// TwinCAT 3 PLC project Untitled1
// ProgramVersion: 3.1.4024.0
// libraries:
//   JSC_MC_Lib, * (Jenny Science AG)
//   JS_MC_REF, * (Jenny Science AG)
//   Sei_Standard, * (Sorenson Engineering)
//   Tc2_MC2, * (Beckhoff Automation GmbH)
//   Tc2_Standard, * (Beckhoff Automation GmbH)
//   Tc2_System, * (Beckhoff Automation GmbH)
//   Tc3_EventLogger, * (Beckhoff Automation GmbH)
//   Tc3_Module, * (Beckhoff Automation GmbH)
// project tree:
//   DUTs/ E_CIM_ERROR_CODES.TcDUT, ST_CONTACT_AFS_PARAMS.TcDUT, ST_CYCLE_TRACKING.TcDUT, ST_ERROR_LOG.TcDUT, ST_JOB_INFO.TcDUT, ST_PLACEMENT_DATA.TcDUT, ST_PLACEMENT_ERROR_INFO.TcDUT, ST_PRODUCTION_DATA.TcDUT, ST_RECIPE_VARS.TcDUT, ST_RFID_DATA.TcDUT, ST_SEARCH_SHAPE.TcDUT
//   GVLs/ GVL.TcGVL
//   ITFs/ ITF_Error.TcIO
//   / PlcTask.TcTTO
//   POUs/00_Shared/ FB_AlarmListener.TcPOU
//   POUs/ FB_AxisBase.TcPOU, FB_Button.TcPOU, FB_Light.TcPOU, FB_Motor.TcPOU, FB_XenaxAxisForceFeedback.TcPOU, MAIN.TcPOU
// real-time tasks:
//   TASK PlcTask: cycle T#10ms, priority 20, ADS port 350
// motion (NC):
//   TASK NC-Task 1 SAF: cycle T#1ms, priority 4, ADS port 501
//   TASK NC-Task 1 SVB: cycle T#10ms, priority 8, ADS port 511
//   AXIS Axis 1 (id 1)
//     General: UnitName=Degree
//     Dynamic: Acceleration=12748, Deceleration=500000, Jerk=382440
//     Velo: RefSync=50, SlowManual=90, FastManual=500, Fast=8498, Maximum=14400
//     PositionAreaControl: Enable=false
//     TargetPosControl: Enable=false
//     OtherSettings: AllowMotionCmdToSlave=true
//     encoder EncType=19
//       EncPara: ScaleFactorNumerator=360, ScaleFactorDenominator=120000, MaxCount=#xffffffff
//         SoftEndMinControl: Range=-29
//         SoftEndMaxControl: Range=29
//     drive DrvType=16
//       DrvPara: MaxCount=#xffffffff, DriveControlDWord=#x00000100
//         Analog: VeloReferenz=14400, VeloScale=32, TorqueSetpointScale=10, ScaleFactorActTorque=0.1
//         TimeComp: TaskDelayCycles=1
//     controller CtrType=9
//       CtrPara: PriorControlFactor=1
//         PosDiffControl: Enable=false, Range=8
//         Observer: BandWidth=20
// I/O:
//   DEVICE Device 2 (EtherCAT), AmsNetId 169.254.194.147.3.1
//     Term 6 (EK1100) [EK1100 EtherCAT Coupler (2A E-Bus)]
//       Term 7 (EL3174) [EL3174 4Ch. Ana. Input +/-10V Diff., +/-20mA SingleEnded, 16 Bit]
//       Term 8 (EL2828) [EL2828 8Ch. Dig. Output 24V, 2A]
//       Term 9 (EL6224) [EL6224 (IO Link Master)]
//       Term 11 (EL9011) [EL9011 End Terminal]
//     Drive 10 (Xvi) [XENAX Xvi 48V8]
// variable links:
//   NC-Task 1 SAF/Axes/Axis 1 <-> Device 2 (EtherCAT)/Drive 10 (Xvi)
//     Drive/Inputs/In/nDataIn1 <-> TxPDO 1/Following Error Actual Value
//     Drive/Inputs/In/nState1 <-> TxPDO 1/Statusword
//     Drive/Inputs/In/nState2 <-> TxPDO 1/Statusword @bit 8
//     Drive/Inputs/In/nState4 @bit 1 <-> WcState/InputToggle
//     Drive/Inputs/In/nState4 <-> WcState/WcState
//     Drive/Outputs/Out/nCtrl1 <-> RxPDO 1/Controlword
//     Drive/Outputs/Out/nCtrl2 <-> RxPDO 1/Controlword @bit 8
//     Drive/Outputs/Out/nDataOut1 <-> RxPDO 1/Target Position
//     Enc/Inputs/In/nDataIn1 <-> TxPDO 1/Position Actual Value
//     Enc/Inputs/In/nState4 @bit 1 <-> WcState/InputToggle
//     Enc/Inputs/In/nState4 <-> WcState/WcState
//   Untitled1/Untitled1 Instance <-> Device 2 (EtherCAT)/Drive 10 (Xvi)
//     PlcTask Inputs/MAIN.motor.ThisMotor.instJS_MC_Init.RxPDO/bWcState <-> WcState/WcState
//     PlcTask Inputs/MAIN.motor.ThisMotor.instJS_MC_Init.RxPDO/diProcessStatusRegister_I2006 <-> TxPDO 2/Process Status Register
//     PlcTask Inputs/MAIN.motor.ThisMotor.instJS_MC_Init.RxPDO/uiStatusword_I6041 <-> TxPDO 2/Statusword
//     PlcTask Inputs/MAIN.motor.ThisMotor.instJS_MC_Init.stSlaveAmsAddr/netId <-> InfoData/AdsAddr/netId
//     PlcTask Inputs/MAIN.motor.ThisMotor.instJS_MC_Init.stSlaveAmsAddr/port <-> InfoData/AdsAddr/port
//   Untitled1/Untitled1 Instance <-> Device 2 (EtherCAT)/Term 6 (EK1100)/Term 9 (EL6224)
//     PlcTask Inputs/MAIN.motor.button.byButtonInput <-> IO-Link Port2/Port2: process data
//     PlcTask Outputs/MAIN.motor.button.byButtonLight <-> IO-Link Port3/Port3: process data
//     PlcTask Outputs/MAIN.motor.light.bAnimationMode <-> IO-Link Port1/Animation Type
//     PlcTask Outputs/MAIN.motor.light.bColor1 <-> IO-Link Port1/Color 1
//     PlcTask Outputs/MAIN.motor.light.bColor2 <-> IO-Link Port1/Color 2
//     PlcTask Outputs/MAIN.motor.light.bColor1Intensity <-> IO-Link Port1/Color 1 Intensity
//     PlcTask Outputs/MAIN.motor.light.bColor2Intensity <-> IO-Link Port1/Color 2 Intensity
//     PlcTask Outputs/MAIN.motor.light.bFlashRate <-> IO-Link Port1/Color Flash Rate (Hz)
//     PlcTask Outputs/MAIN.motor.light.bRotationalMode <-> IO-Link Port1/Rotation Direction
//   Untitled1/Untitled1 Instance <-> NC-Task 1 SAF/Axes/Axis 1
//     PlcTask Inputs/MAIN.motor.ThisMotor.instJS_MC_Init.IS.AxisRef.NcToPlc <-> Outputs/ToPlc
//     PlcTask Outputs/MAIN.motor.ThisMotor.instJS_MC_Init.IS.AxisRef.PlcToNc <-> Inputs/FromPlc

CONFIGURATION Untitled1
    RESOURCE PLC ON TwinCAT3
        TASK PlcTask(INTERVAL := T#10ms, PRIORITY := 20);
        PROGRAM MAIN WITH PlcTask : MAIN;
    END_RESOURCE
END_CONFIGURATION

// ---- DUTs/E_CIM_ERROR_CODES.TcDUT
{attribute 'qualified_only'}
{attribute 'strict'}
TYPE E_CIM_ERROR_CODES :
(
	None := 0,
	//MAIN Errors
	EStopDepressed := 1000,
	//Contact AFS Errors (3000s)
	ContactAFS_SequencerNotOpen := 3001,
	ContactAFS_SequencerDidNotReachPickupPosition := 3002,
	ContactAFS_VibrationTimedOut := 3003
	
);
END_TYPE

// ---- DUTs/ST_CONTACT_AFS_PARAMS.TcDUT
TYPE ST_CONTACT_AFS_PARAMS :
STRUCT
// Keyence Sensor Setpoints                     	     							
	TrackSensorHigh:								INT;
	TrackSensorLow:									INT;
//Vibratory Settings                            	
	TrackAmplitude:									REAL;
//	BowlAmplitude:									REAL;
	BowlOnDelay:									INT;
	BowlOffDelay:									INT;
//Time Delays                                   	
	PartLoadDelay:									INT;
END_STRUCT
END_TYPE

// ---- DUTs/ST_CYCLE_TRACKING.TcDUT
TYPE ST_CYCLE_TRACKING :
STRUCT
	sComponentName:			STRING;
	nCurrentCycles:			UDINT;
	sMaintenance:			STRING;
	nMaxCycles:				UDINT;
END_STRUCT
END_TYPE

// ---- DUTs/ST_ERROR_LOG.TcDUT
TYPE ST_ERROR_LOG :
STRUCT
	sTimeOfError:					STRING;
	eErrorCode:						E_CIM_ERROR_CODES;
//	bErrorCleared:					BOOL;
END_STRUCT
END_TYPE

// ---- DUTs/ST_JOB_INFO.TcDUT
TYPE ST_JOB_INFO :
STRUCT
	sPartNumber:	T_MaxString;
	sRevision:		T_MaxString;
	sJobNumber:		T_MaxString;
END_STRUCT
END_TYPE

// ---- DUTs/ST_PLACEMENT_DATA.TcDUT
TYPE ST_PLACEMENT_DATA :
STRUCT
	nRowCount			:	INT;
	dnColumnCount		:	DINT;
	nHoleCount			:	INT;
	lrXPosition			:	LREAL;
	lrYPosition			:	LREAL;
	lrZPosition			:	LREAL;
	lrZForce			:	LREAL;
	lrXOffset			:	LREAL;
	lrYOffset			:	LREAL;
	lrInsertionFinalZPos:	LREAL;
END_STRUCT
END_TYPE

// ---- DUTs/ST_PLACEMENT_ERROR_INFO.TcDUT
TYPE ST_PLACEMENT_ERROR_INFO :
STRUCT
	stShellNumber:			STRING;
	stContactNumber:		STRING;
	stInsertionErrorInfo:	STRING;
END_STRUCT
END_TYPE

// ---- DUTs/ST_PRODUCTION_DATA.TcDUT
TYPE ST_PRODUCTION_DATA :
STRUCT
	udiPartCount :			UDINT;
	rTenMinuteEfficiency :	REAL;
	tsTime :				TIMESTRUCT;
END_STRUCT
END_TYPE

// ---- DUTs/ST_RECIPE_VARS.TcDUT
TYPE ST_RECIPE_VARS :
STRUCT
	// Recipe Information
	sRecipeName:							STRING;
	//AFS Module Recipe GVL VARS
	//VISION
	lrAreaThreshold:						LREAL := 310000;
	bSwitchSign:							BOOL;
	TopPoint: 								REAL := 960;
	MidPoint: 								REAL := 1225;
	BotPoint: 								REAL := 1600;
	
	//Contact Load Recipe GVL VARS
	//VISION
	aSearchCenterPoint			: TcVnPoint2_REAL;
	aSearchSize					: TcVnPoint2_REAL;
	
	aInnerPointBentPinBottom	: TcVnPoint2_REAL := [650, 550];
	nInnerPointYCamOffsetBottom	: INT := 100;
	aOuterPoint1BentPinBottom	: TcVnPoint2_REAL := [200, 550];
	nOuterPoint1YCamOffsetBottom: INT := 100;
	aOuterPoint2BentPinBottom	: TcVnPoint2_REAL := [650, 100];
	nOuterPoint2YCamOffsetBottom: INT := 100;
	aOuterPoint3BentPinBottom	: TcVnPoint2_REAL := [200, 100];
	nOuterPoint3YCamOffsetBottom: INT := 100;
	aInnerPointEndEffector		: TcVnPoint2_REAL := [800, 470];
	aOuterPoint1EndEffector		: TcVnPoint2_REAL := [200, 470];
	aOuterPoint2EndEffector		: TcVnPoint2_REAL := [800, 100];
	aOuterPoint3EndEffector		: TcVnPoint2_REAL := [200, 100];
	nCamOffsetx					: INT := 72;
	nCamOffsetY					: INT := 12;
	lrBrightnessSensitivy		: LREAL := 16;
	nNumOfHolesThatCanMiss		: INT := 5;
	
	//Pick and Place Recipe Vars
	nNumOfHoles					: INT := 26;
	nRowCount					: INT := 5;
	nNumofShells				: INT := 25;
	lrPnPPreInsertionPos		: LREAL := 78.0;
	lrPnPFinalInsertionPos		: LREAL := 89.719; // Ideal for 26 contact Shell: 89.719;
	lrLocateHolesPos			: LREAL := 77.839;
	nCalibrationImageNum		: INT := 0;
	lrHandoffPosition			: LREAL := 79.5;
	lrInsertionForceThreshold	: LREAL := 1.5;
	lrInsertionStopForce		: LREAL := 0.29;
	lrPinToShoulderLength		: LREAL;
	//Pallet Recipe Vars
	nColumnCount				: INT := 5;
	nPresetPalletNum			: INT := 0;

END_STRUCT

END_TYPE

// ---- DUTs/ST_RFID_DATA.TcDUT
TYPE ST_RFID_DATA :
STRUCT
	aRFIDData:		ARRAY[1..8] OF USINT;
	nPalletID:		UDINT;
	sRecipeName:	STRING;
END_STRUCT
END_TYPE

// ---- DUTs/ST_SEARCH_SHAPE.TcDUT
TYPE ST_SEARCH_SHAPE :
STRUCT
	aCenterPoint			: TcVnPoint2_REAL;
	nHeight					: REAL;
	nWidth					: REAL;
END_STRUCT
END_TYPE

// ---- GVLs/GVL.TcGVL
{attribute 'qualified_only'}
VAR_GLOBAL CONSTANT
	gc_sMachineName:						STRING := 'INVADER CIM';
END_VAR
VAR_GLOBAL
//	GloballrXAxisOverride AT %Q*:			LREAL;
	bAckError:								BOOL;
	eErrorCode:								E_CIM_ERROR_CODES;
	
	gv_uc_bEStopDepressed AT %I*:			BOOL;
	
	bPalletReady:							BOOL;
	bPnPDone:								BOOL;
	bRun:									BOOL;
	bDoorSensorsOK:							BOOL;
	bCurrentIsZero:							BOOL;
	bEStopsOK:								BOOL;
	
	bCameraStart:							BOOL;
	bAutoCalibCamera:						BOOL;
	bContourGeneratorStart:					BOOL;
	bContourCheckStart:						BOOL;
	bEdgeDetectionStart:					BOOL;
	bPass:									BOOL;
	bAFSPartDamaged:						BOOL;
	SequencerJamDetected:					BOOL;
	PnPClear:								BOOL;
	bHMITriggerIncorrectRecipeMessage:		BOOL;
	AttemptingToUnjamSequencer:				BOOL;
	CFReadyForPart:							BOOL;
	CFDamagedPartReceived:					BOOL;
	ResetCFState:							BOOL;
	
	bImageTaken:							BOOL;
	bPalletImagePosition:					BOOL;
	PalletFinished:							BOOL;
	bHMISwapEndEffector:					BOOL;
	bSwapEndEffector:						BOOL;
	//GVs 4 ContactFeedModule
	bCameraStartCF_X:						BOOL;
	bCameraStartCF_Y:						BOOL;
	bCameraDoneCF_X:						BOOL;
	bCameraDoneCF_Y:						BOOL;
	bCalibrateModeCF:						BOOL;
	bInspectModeCF:							BOOL;
	bSetupModeCF:							BOOL;
	bInspectTopCF:							BOOL;
	bContactFailCF:							BOOL;
	rEndEffectorPosCF_X:					REAL;
	rEndEffectorPosCF_Y:					REAL;
	rEndEffectorAngleCF_X:					REAL;
	rEndEffectorAngleCF_Y:					REAL;
	rContactTopPosCF_X:						REAL;
	rContactTopPosCF_Y:						REAL;
	rContactBottomPosCF_X:					REAL;
	rContactBottomPosCF_Y:					REAL;
	rContactAngleCF_X:						REAL;
	rContactAngleCF_Y:						REAL;
	rContactBottomAngleCF_X:				REAL;
	rContactBottomAngleCF_Y:				REAL;
	nBentFail_CF:							INT;
	nOrientFail_CF:							INT;
	rSpatialResolution_CF_X:				REAL;
	rSpatialResolution_CF_Y:				REAL;
	rMaxAngleDeviation_CF: 					REAL := 5.0;
	rHeightOffset:							REAL;
	
	aPointWorld:							ARRAY [0.. 280] OF TcVnPoint3_LREAL;
	bMovePalletToHole:						BOOL;
	nNumOfHoles:							DINT;
	
	bCalibrateModePnP:						BOOL;
	
	bStartPinInspection						:BOOL;
	nCurrentHole							:INT;
	bStartHoleUpdater						:BOOL;
	
	// RECIPE VARS
	stRecipeVars							:ST_RECIPE_VARS;
	stJobInfo:								ST_JOB_INFO;
		
	nCurrentShellNum:						INT;
	aArrayOfPalletIndex0						:ARRAY [1..25] OF INT := [21,22,23,24,25,
																	  16,17,18,19,20,
																	  11,12,13,14,15,
																	  6, 7, 8 , 9,10,
																	  1, 2, 3, 4, 5];

	aArrayOfPalletIndex1						:ARRAY [1..25] OF INT := [7,8,9, 4,5,6,1,2,3];
	aArrayOfPalletIndex							:ARRAY [1..25] OF INT;

	aBentPinz								:ARRAY[1..25] OF ARRAY[1..280] OF INT;
	bStopper								:BOOL;

	
	bErrorState:							BOOL;
	bDisplayInitHoles:						BOOL;
	bMovePalletToOne:						BOOL;
	bTakeCalibImage:						BOOL;
	bGettingPalletToZero:					BOOL;
	
	bRunCalibration:						BOOL;
	bStoreCalibResults:						BOOL;
	bSaveMotorPos:							BOOL;
	aEndEffectorPos:						ARRAY [0..1] OF LREAL;
	aCamZeroPos:							ARRAY [0..1] OF LREAL;
	
	//aCameraToEffectorOffset:				ARRAY [0..1] OF LREAL;
	uiPNPBacklight:							UINT;
	uiPNPBacklightCurrValue:				UINT;
	nNumOfShellsSkipped:					INT := 0;
	
	// Searchbox Settings for Contact Setup
	aCenterPoint			: TcVnPoint2_REAL;
	rWidth					: REAL;
	rHeight					: REAL;
	
	//CAMERA PRIORITY VARS
	bCF_GO:BOOL;
	bAFS_GO:BOOL;
	bPNPWaiting:BOOL;
	bPNP_GO:BOOL;
	bCFWaiting:BOOL;
	
	bHMIAcknowledge : BOOL; 
	
	bPalletStarted : BOOL;
END_VAR
VAR_GLOBAL PERSISTENT
	astCycleTracking:						ARRAY[1..7] OF ST_CYCLE_TRACKING;
	atMaintenanceTimestamp:					ARRAY[1..3] OF LTIME;
	astPlacementErrorInfo:					ARRAY [1..650] OF ST_PLACEMENT_ERROR_INFO;
	nPlacementErrorIndex:					INT := 1;
	astRFIDData:							ARRAY[1..100000] OF ST_RFID_DATA;
END_VAR

// ---- ITFs/ITF_Error.TcIO
INTERFACE ITF_Error

PROPERTY pAckError : BOOL
GET
END_GET
SET
END_SET
END_PROPERTY

PROPERTY pError : BOOL
GET
END_GET
SET
END_SET
END_PROPERTY

PROPERTY pErrorCode : udint
GET
END_GET
SET
END_SET
END_PROPERTY

PROPERTY pErrorDescription : T_MaxString
GET
END_GET
SET
END_SET
END_PROPERTY

END_INTERFACE

// ---- POUs/MAIN.TcPOU
PROGRAM MAIN

// MOTOR WITH LIGHT AND BUTTON BRANCH

VAR	
	// array to be passed to the FB_Motor
	aTargets : ARRAY[1..10] OF INT := [0, 360, 720, 0, 720, -720, 0, -360, 360, 0];
	
	motor : FB_Motor;
	//light : FB_Light;
	
	init : BOOL := TRUE;
END_VAR

IF init THEN
	motor.mInitialize(aInputArray := aTargets);
	init := FALSE;
END_IF

// Call the FB to run the motors functions
//motor.mStates();
motor();

END_PROGRAM

// ---- POUs/FB_Motor.TcPOU
FUNCTION_BLOCK FB_Motor

VAR
	aInputTargets : ARRAY[1..10] OF INT;	

	ThisMotor : FB_XenaxAxisForceFeedback;
	motorParameters : ST_MOTION_PARAMS;
	
	// Movement states for the motor
	enumStates : (INITIALIZE_VALUES, INITIALIZE, MOVING, WAIT, GET_NEXT_TARGET, MOVE_TO_TARGET);
	nEnumIndex : INT := 0;
	aEnumStates : ARRAY[1..6] OF INT := [12, 1, 0, 2, 3, 6];
	(*	
		enumStates	| INITIALIZE_VALUES | INITIALIZE | MOVING | WAIT | GET_NEXT_TARGET | MOVE_TO_TARGET |
		aEnumStates |          12		| 	  1		 |    0	  |   2  |        3		   |        6       |
		Color		|		 white      |    red     |  green |orange|	   yellow      |      cyan		|
	
		The colors are parallel to the state the motor is in
	*)
	light : FB_Light;
	button : FB_Button;
	bButton : BOOL;
	
	tonLightFlashDelay : TON := (PT := T#600MS);
	bFlashState : BOOL;
	
END_VAR

bButton := button.byButtonInput; // set bool from the state of the button
button.mButtonLight(); // light for the button if it is pressed

IF bButton THEN
	mStates(); // keep running through states
// ^^ could have manager to have a stack to follow commands
// but for this purpose, its ok

ELSE
	// set the color to red
	light.mSetColor(nInputNumber := 1);
	
	IF bFlashState THEN // light is on
		tonLightFlashDelay(IN := TRUE);
		// check if time has elapsed
		IF tonLightFlashDelay.Q THEN
			// turn the light off
			light.mSetAnimation(0);
			// set bFlashState to FALSE
			bFlashState := FALSE;
			// reset timer
			tonLightFlashDelay(IN := FALSE);
		END_IF
		
	ELSE // light is off
		tonLightFlashDelay(IN := TRUE);
		// check if time has elapsed
		IF tonLightFlashDelay.Q THEN
			// turn the light on
			light.mSetAnimation(1);
			// set bFlashState to TRUE
			bFlashState := TRUE;
			// reset timer
			tonLightFlashDelay(IN := FALSE);
		END_IF
	
	END_IF
	

END_IF

METHOD mInitialize : BOOL

VAR_INPUT
	aInputArray : ARRAY[1..10] OF INT;
END_VAR
aInputTargets := aInputArray;
END_METHOD

METHOD mStates : BOOL

VAR_INPUT
END_VAR

VAR_INST
	// Track index location of input array & value at current index of input array
	nTargetIndex : INT := 1;
	nTargetValue : INT := 0;
	
	
	// Wait timer between move commands
	tonWaitTimer : TON := (PT := T#500MS);
END_VAR
Thismotor(usiRefernceDirection := INT_TO_USINT(E_JS_MC_REF_MODE.Positive));
light.mSetAnimation(bInputValue := 1);

CASE enumStates OF
	INITIALIZE_VALUES:
		nEnumIndex := 1;
		light.mSetColor(nInputNumber := nEnumIndex);
		
		motorParameters.TargetPos := 0;
		motorParameters.Jerk := 20000;
		motorParameters.TargetAccel := 2000;
		motorParameters.TargetDecel := 2000;
		motorParameters.TargetVel := 1000;
		enumStates := INITIALIZE;
		
		
	INITIALIZE:
		nEnumIndex := 2;
		light.mSetColor(nInputNumber := nEnumIndex);
		
		ThisMotor.Initialize(TRUE);
		IF ThisMotor.DidInitialize THEN
			nTargetValue := 0;
			enumStates := MOVE_TO_TARGET;
		END_IF
		
		
	MOVING:
		nEnumIndex := 3;
		light.mSetColor(nInputNumber := nEnumIndex);
		
		ThisMotor.MoveAbs(Execute := TRUE, MotionParams := motorParameters);
		IF ThisMotor.DidMoveAbs THEN
			ThisMotor.MoveAbs(Execute := FALSE, MotionParams := motorParameters);
			enumStates := WAIT;
		END_IF
		
		
	WAIT:
		nEnumIndex := 4;
		light.mSetColor(nInputNumber := nEnumIndex);
		
		tonWaitTimer(IN := TRUE);
		
		IF tonWaitTimer.Q THEN
			tonWaitTimer(IN := FALSE);
			enumStates := GET_NEXT_TARGET;
		END_IF

		
	GET_NEXT_TARGET:
		nEnumIndex := 5;
		light.mSetColor(nInputNumber := nEnumIndex);
		
		IF nTargetIndex + 1 > UINT_TO_INT(SIZEOF(aInputTargets)/2) THEN // divide by 2 since the array type is of int (2 bytes per entry)
			nTargetIndex := 1;
		END_IF

		nTargetValue := aInputTargets[nTargetIndex];
		
		nTargetIndex := nTargetIndex + 1;
		
		enumStates := MOVE_TO_TARGET;
		
		
	MOVE_TO_TARGET:
		nEnumIndex := 6;
		light.mSetColor(nInputNumber := nEnumIndex);
		
		motorParameters.TargetPos := nTargetValue;
		enumStates := MOVING;
		
END_CASE
END_METHOD

END_FUNCTION_BLOCK

// ---- POUs/FB_XenaxAxisForceFeedback.TcPOU
(* 
:WARNING: Still in development

:Description: This function block should be used to control a jenny science axis

:Instructions for use:

	- Update this function block every cycle
	
Version history:

+-------------+------------+----------------+--------+---------------+------------------------------------------+
|Date         | Version    | created under  | Author |Checked By     | Remark                                   |
+=============+============+================+========+===============+==========================================+
|10-11-2019   | 0.0.0      | V3.1.4022.28   | C.B.   |               | 								            |
+-------------+------------+----------------+--------+---------------+------------------------------------------+

*)

FUNCTION_BLOCK FB_XenaxAxisForceFeedback EXTENDS FB_AxisBase
VAR_INPUT 
	usiRefernceDirection				: USINT;
END_VAR
VAR
(* Axis *)
	instJS_MC_Init						: JS_MC_Init; //create PLC axis link through this FB instead of traditional AXIS_REF
(* JSCM_Mc_Lib *)
	instJS_MC_Power 					: JS_MC_Power;
	instJS_MC_Reference 				: JS_MC_Reference;
	instJS_MC_ReadAxisError				: JS_MC_ReadAxisError;
	instJS_MC_ReadStatus 				: JS_MC_ReadStatus;
	instJS_MC_Reset 					: JS_MC_Reset;
	instJS_MC_CyclicIn 					: JS_MC_CyclicIn;
	instJS_MC_ForceCalibration			: JS_MC_ForceCalibration;
	instJS_MC_CyclicOut 				: JS_MC_CyclicOut;
	instJS_MC_ReadPSR					: JS_MC_ReadPSR;
	instJS_MC_ReadActualPosition		: JS_MC_ReadActualPosition;
(* Internal Vars *)
	bCyclic:							BOOL;
	bInit:								BOOL := TRUE; //intialize on first plc cycle 
	CommunicationError:					BOOL;
	GetForceAtFailure:					LREAL;
(* Property Variables *)
	bValid:								BOOL;
END_VAR

(*
	Axis FB speciific to jenny science drive. Provides the necessary cyclic communication for JS_MC_Lib and the use of force feed back.
*)
//Calls all motion blocks cyclically
JsCyclicComm();
CyclicComm();

PROPERTY ActAccl : LREAL
GET
ActAccl := CalculateAccl();
END_GET
END_PROPERTY

PROPERTY ActForce : lreal
GET
ActForce := ABS((DINT_TO_LREAL(instJS_MC_Init.RxPDO.diI_ForceActual_I2005))/1000);
END_GET
END_PROPERTY

PROPERTY ActPos : lreal
GET
//Scaled to millimeters 
ActPos := (DINT_TO_LREAL(instJS_MC_Init.RxPDO.diPositionActualValue_I6064))/1000;
END_GET
END_PROPERTY

METHOD Axis_PowerOff : BOOL
VAR_INPUT
	Execute:		BOOL;
END_VAR
VAR_INST
	PowerState:		INT;
	rtrigExecutePower :	R_TRIG;
END_VAR
CASE PowerState OF

	0: 	
		rtrigExecutePower(CLK := Execute);
		IF rtrigExecutePower.Q THEN
			Axis_PowerOff := FALSE;
			bDidPowerOff := FALSE;
			bDidInitialize := FALSE;
			PowerState := 10;
		END_IF
			
	10:
		IF instJS_MC_Power.Status THEN		
			instJS_MC_Power.Enable := FALSE;										 
  			instJS_MC_Power.Enable_Positive := 	FALSE;																	
  			instJS_MC_Power.Enable_Negative	:= FALSE;										
  			instJS_MC_Power.Override := 0;												
		ELSIF NOT instJS_MC_Power.Status THEN
			Axis_PowerOff := TRUE;
			bDidPowerOff := TRUE;
			PowerState := 0;
		END_IF
END_CASE
END_METHOD

METHOD Axis_PowerOn : BOOL
VAR_INPUT
	Execute:				BOOL;
END_VAR
VAR_INST
	State:					INT;
	fbTimer:				TON;
END_VAR
rtrigExecute(CLK := Execute);
CASE State OF
	0:  //Exectue	
		IF rtrigExecute.Q THEN
			Axis_PowerOn := FALSE;
			bDidPowerOn := FALSE;
			State := 5;
		END_IF
	5: //Cyclic valid
		IF instJS_MC_CyclicIn.Valid THEN
			State := 10;
		END_IF
	10: //Reset 
		instJS_MC_Reset.Execute := TRUE;
		State := 20;
	20: //reset done 
		IF instJS_MC_Reset.Done THEN
			instJS_MC_Reset.Execute := FALSE;
			State := 25;
		END_IF
	
	25:
		instJS_MC_Power.Enable_Positive := 	FALSE;							
  		instJS_MC_Power.Enable_Negative := 	FALSE;
		instJS_MC_Power.Enable := FALSE;
		State := 30;
		
	30: //Enable
		instJS_MC_Power.Enable_Positive := 	TRUE;		(* Advance movement enable in positive direction *)									
  		instJS_MC_Power.Enable_Negative := 	TRUE;		(* Advance movement enable in negative direction *)	
  		instJS_MC_Power.Override	:= 100;	
		instJS_MC_Power.Enable := TRUE;
		IF instJS_MC_Power.Status THEN
			State := 40;
		ELSE
			fbTimer(IN:= TRUE, PT:= T#1S);
			IF fbTimer.Q THEN
				fbTimer(IN := FALSE);
				State := 10;
			END_IF
		END_IF	
		
	40: //Delay time
		fbTimer(IN := TRUE, PT:= T#1S);
		IF fbTimer.Q THEN
			fbTimer(IN := FALSE);
			Axis_PowerOn := TRUE;
			bDidPowerOn := TRUE;
			State := 0;
		END_IF
END_CASE
END_METHOD

METHOD CalculateAccl : LREAL
VAR_INST 
	PrevVelo: 		LREAL;
	CurrentVelo: 	LREAL;
END_VAR
(*
 Estimated the actual accleration based on the rate of change of velocity
*)
PrevVelo := CurrentVelo;
CurrentVelo := ActVelo;
CalculateAccl := (CurrentVelo - PrevVelo)/0.001;
END_METHOD

METHOD Calibrate : BOOL
VAR_INPUT
	Execute	: 						BOOL;
	StartPosition :					LREAL;	// in millimeters 
	EndPosition:					LREAL; // in millimeters 
	ZeroPreviousForceData:			BOOL;
END_VAR

VAR_INST
	State:					INT;
	rtrigExecute:			R_TRIG;
END_VAR
CASE State OF
	0: 	// Execute
		rtrigExecute(CLK := Execute);
		IF rtrigExecute.Q THEN
			Calibrate := FALSE;
			bBusy := TRUE;
			State := 10;
		END_IF
	10: // Calibrate to start and end positions 
		instJS_MC_ForceCalibration.IterativeFcDisable := ZeroPreviousForceData;
		instJS_MC_ForceCalibration.StartPosition := LREAL_TO_DINT(StartPosition*1000);
		instJS_MC_ForceCalibration.EndPosition := LREAL_TO_DINT(EndPosition*1000);
		instJS_MC_ForceCalibration.Execute := TRUE;	
		State := 20;
	20:
		IF instJS_MC_ForceCalibration.Done THEN
			instJS_MC_ForceCalibration.Execute := FALSE;
			Reset(Execute := FALSE);
			State := 30;
		END_IF
	30: // reset 
		IF Reset(Execute := TRUE) THEN
			Reset(Execute := FALSE);
			Calibrate := TRUE;
			bBusy := FALSE;
			State := 0;
		END_IF 
END_CASE
END_METHOD

METHOD CyclicComm
(*
	This method proves the cyclic communication for all Twincat motion function blocks and the removal of function blocks used from the JS_Mc_Lib
*)
fbMoveAbs1(Axis:= instJS_MC_Init.pstAxis^.AxisRef);
fbMoveAbs2(Axis:= instJS_MC_Init.pstAxis^.AxisRef);
fbMoveAbs3(Axis:= instJS_MC_Init.pstAxis^.AxisRef);
fbHalt(Axis:= instJS_MC_Init.pstAxis^.AxisRef);
//fbStop(Axis:= instJS_MC_Init.pstAxis^.AxisRef);
fbReset(Axis := instJS_MC_Init.pstAxis^.AxisRef);
fbJog(Axis:= instJS_MC_Init.pstAxis^.AxisRef);
fbMoveRel(Axis:= instJS_MC_Init.pstAxis^.AxisRef);
fbMoveVelo(Axis:= instJS_MC_Init.pstAxis^.AxisRef);
fbMoveModulo(Axis:= instJS_MC_Init.pstAxis^.AxisRef);

bError := instJS_MC_ReadAxisError.AxisError;
END_METHOD

PROPERTY ForceAtFailure  : lreal
GET
ForceAtFailure := GetForceAtFailure;
END_GET
END_PROPERTY

METHOD Initialize : BOOL
VAR_INPUT
	Execute:				BOOL;
END_VAR
VAR_INST
	InitState:				INT;
	rtrigInit :				R_TRIG;
	fbTimer:				TON;
END_VAR
CASE InitState OF
	0: 	// Execute
		rtrigInit(CLK := Execute);
		IF rtrigInit.Q THEN
			Initialize := FALSE;
			bDidInitialize := FALSE;
			bBusy := TRUE;
			InitState := 10;
		END_IF
	10: //Power on 
		IF Axis_PowerOn(TRUE) THEN
			Axis_PowerOn(FALSE);
			InitState:= 15;
		END_IF
		
	15: IF instJS_MC_Power.Status THEN
			InitState := 20;
		ELSE
			IF Axis_PowerOff(TRUE) THEN
				Axis_PowerOff(FALSE);
				InitState := 10;
			END_IF
		END_IF
		
	20: //Reference
		IF Ref(TRUE) THEN
			Ref(FALSE);
			InitState := 30;
		END_IF
	30:
		Initialize := TRUE;
		bDidInitialize := TRUE;
		bBusy := FALSE;
		InitState := 0;
END_CASE
END_METHOD

METHOD JsCyclicComm
VAR_INST 
	State:		INT;
END_VAR
(* 
	starts the PLCopen status machine and the communication to the axis device for entering instructions of the cyclic task.
*)

IF bInit THEN 
	instJS_MC_Init.OperationMode := gcJS_MC.jsmcMODE_CYCLIC_SYNC;
	instJS_MC_Init();
	bInit := instJS_MC_Init.Error;
	instJS_MC_Reference.ReferenceMode := usiRefernceDirection; //reference direction 																			 
	instJS_MC_ReadAxisError.Enable := TRUE;
	instJS_MC_ReadStatus.Enable := TRUE;
	instJS_MC_ReadPSR.Enable := TRUE;		
END_IF

IF NOT bInit THEN
	
	CASE State OF 
		0: (* Check communication errors and start cyclic In/Out*)
			IF instJS_MC_CyclicIn.Error THEN				
				bCyclic := FALSE;
				CommunicationError := TRUE;
				state := 10;
			ELSE
				bCyclic := TRUE;
			END_IF	
		10: (* Communication interrupted *)
			instJS_MC_Reset.Execute := FALSE;
			instJS_MC_Reference.Execute := FALSE;
			instJS_MC_Power.Enable := FALSE;
			State := 0;
	END_CASE

	instJS_MC_CyclicIn( pstAxis := instJS_MC_Init.pstAxis, Enable := bCyclic);
	instJS_MC_Init.pstAxis^.AxisRef.ReadStatus();
	instJS_MC_Power(pstAxis:= instJS_MC_Init.pstAxis);
	instJS_MC_Reference(pstAxis := instJS_MC_Init.pstAxis); 					
    instJS_MC_ReadAxisError(pstAxis := instJS_MC_Init.pstAxis);
    instJS_MC_ReadStatus(pstAxis := instJS_MC_Init.pstAxis); 		
    instJS_MC_Reset(pstAxis := instJS_MC_Init.pstAxis); 					
    instJS_MC_ForceCalibration(pstAxis := instJS_MC_Init.pstAxis);	
    instJS_MC_ReadPSR(pstAxis := instJS_MC_Init.pstAxis);		
	instJS_MC_CyclicOut(pstAxis := instJS_MC_Init.pstAxis);	
END_IF
END_METHOD

METHOD PUBLIC MaxForceReset : BOOL
VAR_INPUT
	Execute:			BOOL;
END_VAR
VAR_INST
	State:				INT;
	rtrigHalt:			R_TRIG;
END_VAR
rtrigHalt(CLK := Execute);
CASE State OF 
	0:	//Execute
		IF rtrigHalt.Q THEN
			MaxForceReset := FALSE;
			bDidHalt := FALSE;
			State := 10;
		END_IF
	10:// Reset to update the actual position and confirm again all execute commands to FALSE
		IF Reset(TRUE) THEN
			Reset(FALSE);
			fbHalt.Execute := FALSE;
			fbMoveAbs1.Execute := FALSE;
			fbMoveAbs2.Execute := FALSE;
			fbMoveAbs3.Execute := FALSE;
			fbMoveModulo.Execute := FALSE;
			fbMoveRel.Execute := FALSE;
			fbMoveVelo.Execute := FALSE; 
			State := 20;
		END_IF
	20: //Done 
		MaxForceReset := TRUE;
		bDidHalt := TRUE;
		State := 0;
END_CASE
END_METHOD

METHOD Pause : BOOL
Pause := FALSE;
instJS_MC_Power.Override := 0;
Pause := TRUE;
END_METHOD

METHOD Ref : BOOL
VAR_INPUT
	Execute:	BOOL;
END_VAR
VAR_INST 
	RefState:				INT;
	rtrigRef:				R_TRIG;
END_VAR
CASE RefState OF	
	0: //Execute 
		rtrigRef(CLK := Execute);
		IF rtrigRef.Q THEN
			bDidRef := FALSE;
			Ref := FALSE;
			RefState := 10;
		END_IF
	10: //Check for previous reference 
		IF instJS_MC_ReadPSR.ProcessStatusRegister.bReference THEN
			RefState := 30;
		ELSIF NOT instJS_MC_ReadPSR.ProcessStatusRegister.bReference THEN
			instJS_MC_Reference.Execute := TRUE;
			RefState := 20;
		END_IF
	20: //Wait for ref complete
		IF instJS_MC_Reference.Done THEN
			instJS_MC_Reference.Execute := FALSE;
			RefState := 30;
		END_IF
	30: 
		bDidRef := TRUE;
		Ref := TRUE;
		RefState := 0;
END_CASE
END_METHOD

METHOD Resume : BOOL
VAR_INPUT
	ResumeOverride: LREAL;
END_VAR
Resume := FALSE;
instJS_MC_Power.Override := ResumeOverride;
Resume := TRUE;
END_METHOD

METHOD SetAxisOverride
VAR_INPUT
	Override:				UDINT;						//Set value from 0-100%
END_VAR
(*
	This method passes an override value to the NC 
*)
instJS_MC_Power.Override := Override;
END_METHOD

END_FUNCTION_BLOCK

// ---- POUs/FB_AxisBase.TcPOU
(* 
:WARNING: Still in development

:Description: This function block should be used to control a basic servo axis.

:Instructions for use:

	- Update this function block every cycle
	
Version history:

+-------------+------------+----------------+--------+---------------+------------------------------------------+
|Date         | Version    | created under  | Author |Checked By     | Remark                                   |
+=============+============+================+========+===============+==========================================+
|10-11-2019   | 0.0.0      | V3.1.4022.28   | C.B.   |               | 								            |
+-------------+------------+----------------+--------+---------------+------------------------------------------+

*)

FUNCTION_BLOCK FB_AxisBase IMPLEMENTS ITF_Error
VAR_INPUT
END_VAR
VAR
(* Axis Ref *)
	Axis:						AXIS_REF;
(* FB's *)
	fbMoveRel:					MC_MoveRelative;
	fbMoveAbs1:				 	MC_MoveAbsolute;
	fbMoveAbs2:					MC_MoveAbsolute;
	fbMoveAbs3:					MC_MoveAbsolute;
	fbMoveVelo:					MC_MoveVelocity;
	fbMoveModulo:				MC_MoveModulo;
	fbJog:						MC_Jog;
	fbReset:		 			MC_Reset;
	fbPower: 					MC_Power;
	fbHalt:						MC_Halt;
	fbHome:						MC_Home;
	fbStop:						MC_Stop;
(* Axis Monitoring *)
	stParameterSet :			ST_AxisParameterSet;
	fbReadParameterSet :		MC_ReadParameterSet;
	fbWriteParameterSet :		MC_WriteParameter;
(* Event based POUs/Vars*)
	fbTcAlarm_Error:			FB_TcAlarm;
	fbAlarmListener:			FB_AlarmListener;
	stSeiEvents:				ST_Sei_Events;
	fbTcEventLogger:			FB_TcEventLogger;
	bAlarmCleared:				BOOL;
(* Property Variables*)
	bClearError:				BOOL;
	bAckError:					BOOL;
	bError:						BOOL;
	udnErrorCode:				UDINT;
	bBusy:						BOOL;
	bActive:					BOOL;
	bStatus:					BOOL;
	sErrorDescription:			T_MaxString;
	bAborted:					BOOL;
	bDidRef:					BOOL;
	bDidInitialize:				BOOL;
	bDidMoveAbs:				BOOL;
	bDidMoveMod:				BOOL;
	bDidMoveRel:				BOOL;
	bDidReset:					BOOL;
	bDidPowerOff:				BOOL;
	bDidPowerOn:				BOOL;
	bDidMoveVelo:				BOOL;
	bDidHalt:					BOOL;
	bDidZero:					BOOL;
	bErrorConfirmed:			BOOL;
	
(*Utility*)
	rtrigExecute:				R_TRIG;
END_VAR

//Calls all motion blocks cyclically
CyclicComm();

PROPERTY Aborted : BOOL
GET
Aborted := bAborted;
END_GET
END_PROPERTY

PROPERTY ActAccl : LREAL
GET
ActAccl := Axis.NcToPlc.ActAcc;
END_GET
END_PROPERTY

PROPERTY Active : BOOL
GET
Active := bActive;
END_GET
END_PROPERTY

PROPERTY ActPos : LREAL
GET
ActPos := Axis.NcToPlc.ActPos;
END_GET
END_PROPERTY

PROPERTY ActVelo : LREAL
GET
ActVelo := Axis.NcToPlc.ActVelo;
END_GET
END_PROPERTY

METHOD Axis_Jog 
VAR_INPUT
	JogParams: 				ST_JOG_PARAMS;
END_VAR
VAR_INST
	State:	INT;
	rtrigExecute :	R_TRIG;
	Timer:				TON;
END_VAR
(*
	This method allows the user to enable an axis for jog. Jog modes are set depending on the user imput of jog distance
*)
 //Jog
(*Incremental Jog*)
	IF JogParams.Distance <> 0 THEN	
		fbJog.Mode := MC_JOGMODE_INCHING; 
		fbJog.Velocity := JogParams.TargetVel; 
		fbJog.Position := JogParams.Distance; 
		fbJog.JogForward := JogParams.JogForward; 
		fbJog.JogBackwards := JogParams.JogBackward; 
		fbJog.Acceleration := JogParams.TargetAccel; 
		fbJog.Deceleration := JogParams.TargetDecel;
		fbJog.Jerk := JogParams.Jerk; 
	END_IF
(*Continuous Jog*)
	IF JogParams.Distance = 0  THEN
		fbJog.Mode := MC_JOGMODE_CONTINOUS;
		fbJog.Velocity := JogParams.TargetVel; 
		fbJog.Position := JogParams.Distance; 
		fbJog.JogForward := JogParams.JogForward; 
		fbJog.JogBackwards := JogParams.JogBackward; 
		fbJog.Acceleration := JogParams.TargetAccel; 
		fbJog.Deceleration := JogParams.TargetDecel; 
		fbJog.Jerk := JogParams.Jerk; 
	END_IF
END_METHOD

METHOD Axis_MoveModulo : BOOL
VAR_INPUT
	Execute:			BOOL;
	MotionParams:		ST_MOTION_PARAMS;
END_VAR
VAR_INST
	State :				INT;
END_VAR
rtrigExecute(CLK := Execute);	
CASE State OF
	0: //Execute 
		IF rtrigExecute.Q THEN
			Axis_MoveModulo := FALSE;
			bDidMoveMod := FALSE;
			State := 10;
		END_IF
	10: //Move modulo 
		fbMoveModulo.Position:= MotionParams.TargetPos; 
		fbMoveModulo.Velocity:= MotionParams.TargetVel; 
		fbMoveModulo.Acceleration:= MotionParams.TargetAccel; 
		fbMoveModulo.Deceleration:= MotionParams.TargetDecel; 
		fbMoveModulo.Jerk:= MotionParams.Jerk; 
		fbMoveModulo.Direction:= MotionParams.Direction; 
		fbMoveModulo.BufferMode:= MotionParams.BufferMode; 
		fbMoveModulo.Execute:= TRUE;
		IF fbMoveModulo.Done THEN
			bDidMoveMod := TRUE;
			fbMoveModulo.Execute := FALSE;
			Axis_MoveModulo := TRUE;
			State := 0;
		END_IF
END_CASE
END_METHOD

METHOD Axis_MoveRelative : BOOL
VAR_INPUT
	Execute:			BOOL;
	MotionParams:		ST_MOTION_PARAMS;
END_VAR
VAR_INST
	State :		INT;
END_VAR
rtrigExecute(CLK := Execute);
CASE State OF	
	0: //Execute
		IF rtrigExecute.Q THEN
			Axis_MoveRelative := FALSE;
			bDidMoveRel := FALSE;
			State := 10;
		END_IF
	10: //Move relative
			fbMoveRel.Execute:= TRUE;
			fbMoveRel.Distance := MotionParams.TargetDistance;
			fbMoveRel.Velocity:= MotionParams.TargetVel; 
			fbMoveRel.Acceleration:= MotionParams.TargetAccel; 
			fbMoveRel.Deceleration:= MotionParams.TargetDecel; 
			fbMoveRel.Jerk:= MotionParams.Jerk; 
		IF fbMoveRel.Done THEN
			fbMoveRel.Execute := FALSE;
			Axis_MoveRelative := TRUE;
			bDidMoveRel := TRUE;
			State := 0;
		END_IF

END_CASE
END_METHOD

METHOD Axis_PowerOff : BOOL
VAR_INPUT
	Execute:	BOOL;
END_VAR
VAR_INST
	State:	INT;
END_VAR
rtrigExecute(CLK := Execute);
CASE State OF
	0: //Execute 
		IF rtrigExecute.Q THEN
			Axis_PowerOff := FALSE;
			bDidPowerOff := FALSE;
			bDidInitialize := FALSE;
			State := 10;
		END_IF	
	10: //Power Off 
		IF fbPower.Status THEN
			fbPower.Enable:= FALSE;
			fbPower.Enable_Positive:= FALSE;
			fbPower.Enable_Negative:= FALSE; 
			fbPower.Override:= 0;
			Axis_PowerOff := FALSE;
		ELSIF NOT fbPower.Status THEN
			Axis_PowerOff := TRUE;
			bDidPowerOff := TRUE;
			State := 0;
		END_IF
END_CASE
END_METHOD

METHOD Axis_PowerOn : BOOL
VAR_INPUT
	Execute:	BOOL;
END_VAR
VAR_INST
	State:	INT;
END_VAR
rtrigExecute(CLK := Execute);
CASE State OF
	0:  //Exectue	
		IF rtrigExecute.Q THEN
			bDidPowerOn := FALSE;
			Axis_PowerOn := FALSE;
			State := 10;
		END_IF
		
	10: //Enable
		fbPower.Enable:= TRUE; 
		fbPower.Enable_Positive:= TRUE; 
		fbPower.Enable_Negative:= TRUE; 
		fbPower.Override:= 100;
		IF fbPower.Status THEN
			Axis_PowerOn := TRUE;
			bDidPowerOn := TRUE;
			State := 0;
		END_IF
END_CASE
END_METHOD

METHOD Axis_Zero : BOOL
VAR_INPUT
	Execute:			BOOL;
	MotionParams:		ST_MOTION_PARAMS;
END_VAR
VAR_INST
	State :				INT;
END_VAR
rtrigExecute(CLK := Execute);	
CASE State OF
	0: //Execute 
		IF rtrigExecute.Q THEN
			Axis_Zero := FALSE;
			bDidZero := FALSE;
			State := 10;
		END_IF
	10: //Home 
		fbHome.Position:= 0; 
		fbHome.HomingMode := MC_HomingMode.MC_Direct;
		fbHome.Execute := TRUE;
		IF fbHome.Done THEN
			bDidZero := TRUE;
			fbHome.Execute := FALSE;
			Axis_Zero := TRUE;
			bDidZero := TRUE;
			State := 0;
		END_IF
END_CASE
END_METHOD

PROPERTY Busy : BOOL
GET
Busy := bBusy;
END_GET
END_PROPERTY

METHOD CyclicComm
(*
	This method proves the cyclic communication for all Twincat motion function blocks
*)
Axis();
fbPower(Axis:= Axis);
fbMoveAbs1(Axis:= Axis);
fbMoveAbs2(Axis:= Axis);
fbMoveAbs3(Axis:= Axis);
fbHalt(Axis:= Axis);
fbStop(Axis:= Axis);
fbReset(Axis := Axis);
fbJog(Axis:= Axis);
fbMoveRel(Axis:= Axis);
fbMoveVelo(Axis:= Axis);
fbMoveModulo(Axis:= Axis);
fbHome(Axis:= Axis);
mErrorMonitoring();
END_METHOD

PROPERTY DidHalt : BOOL
GET
DidHalt := bDidHalt;
END_GET
END_PROPERTY

PROPERTY DidInitialize : BOOL
GET
DidInitialize := bDidInitialize;
END_GET
END_PROPERTY

PROPERTY DidMoveAbs : BOOL
GET
DidMoveAbs := bDidMoveAbs;
END_GET
END_PROPERTY

PROPERTY DidMoveMod : BOOL
GET
DidMoveMod := bDidMoveMod;
END_GET
END_PROPERTY

PROPERTY DidMoveRelative : BOOL
GET
DidMoveRelative := bDidMoveRel;
END_GET
END_PROPERTY

PROPERTY DidMoveVelo : BOOL
GET
DidMoveVelo := bDidMoveVelo;
END_GET
END_PROPERTY

PROPERTY DidPowerOff : BOOL
GET
DidPowerOff := bDidPowerOff;
END_GET
END_PROPERTY

PROPERTY DidPowerOn : BOOL
GET
DidPowerOn := bDidPowerOn;
END_GET
END_PROPERTY

PROPERTY DidRef : BOOL
GET
DidRef := bDidRef;
END_GET
END_PROPERTY

PROPERTY DidReset : BOOL
GET
DidReset := bDidReset;
END_GET
END_PROPERTY

PROPERTY DidZero : BOOL
GET
DidZero := bDidZero;
END_GET
END_PROPERTY

METHOD PUBLIC Halt : BOOL
VAR_INPUT
	Execute:			BOOL;
	MotionParams:		ST_MOTION_PARAMS;
END_VAR
VAR_INST
	State:				INT;
	rtrigHalt:			R_TRIG;
END_VAR
rtrigHalt(CLK := Execute);
CASE State OF 
	0:	//Execute
		IF rtrigHalt.Q THEN
			Halt := FALSE;
			bDidHalt := FALSE;
			State := 10;
		END_IF
	10://Halt 
		fbHalt.Deceleration:= MotionParams.TargetDecel; 
		fbHalt.Jerk:= MotionParams.Jerk; 
		fbHalt.Execute:= TRUE;
		IF fbHalt.Done THEN 
			State := 20;
		END_IF
	20://Confirm halt done and set any execute commands to FALSE
		IF fbHalt.Execute THEN
			fbHalt.Execute := FALSE;
			fbMoveAbs1.Execute := FALSE;
			fbMoveAbs2.Execute := FALSE;
			fbMoveModulo.Execute := FALSE;
			fbMoveRel.Execute := FALSE;
			fbMoveVelo.Execute := FALSE;
			State := 30;
		END_IF
	30:// Reset to update the actual position and confirm again all execute commands to FALSE
		IF Reset(TRUE) THEN
			Reset(FALSE);
			fbHalt.Execute := FALSE;
			fbMoveAbs1.Execute := FALSE;
			fbMoveAbs2.Execute := FALSE;
			fbMoveAbs3.Execute := FALSE;
			fbMoveModulo.Execute := FALSE;
			fbMoveRel.Execute := FALSE;
			fbMoveVelo.Execute := FALSE; 
			State := 40;
		END_IF
	40: //Done 
		Halt := TRUE;
		bDidHalt := TRUE;
		State := 0;
END_CASE
END_METHOD

METHOD Initialize : BOOL
VAR_INPUT
	Execute:		BOOL;
END_VAR
VAR_INST
	State:	INT;
	rtrigInitialize :	R_TRIG;
	Timer:				TON;
END_VAR
rtrigInitialize(CLK := Execute);
CASE State OF	
	0: //Execute  	
		IF rtrigInitialize.Q THEN
			Initialize := FALSE;
			bDidInitialize := FALSE;
			State := 10;
		END_IF
	10 :  // Reset Axis
		IF Reset(TRUE) THEN
			Reset(FALSE);
			State := 20;
		END_IF				
	20 : // Power on axis
		IF Axis_PowerOn(TRUE) THEN
			Axis_PowerOn(FALSE);
			State := 30;
		END_IF
	30: // Dwell Time before calling any third party axis reference if applicable 
		Timer(IN := TRUE, PT := T#2S);
		IF Timer.Q THEN
			Timer(IN := FALSE);
			State := 40;
		END_IF
	40: //Reference axis
		IF Ref(TRUE) THEN 
			Ref(FALSE);
			Initialize := TRUE;
			bDidInitialize := TRUE;
			State := 0;
		END_IF					
END_CASE
END_METHOD

(*
	Error monitoring for MC function blocks
*)
METHOD mErrorMonitoring 
VAR_INST
	bFbError:	BOOL;
	bNcError:	BOOL;
END_VAR
(*Check for Fb error*)
IF fbPower.Error OR 
fbMoveAbs1.Error OR 
fbMoveAbs2.Error OR 
fbMoveAbs3.Error OR
fbHalt.Error OR 
fbReset.Error OR 
fbJog.Error OR 
fbMoveRel.Error OR 
fbMoveVelo.Error OR 
fbMoveModulo.Error THEN
	bFbError := TRUE;
ELSE 
	bFbError := FALSE;
END_IF

(*Get Fb error code*)
IF fbPower.Error THEN
	udnErrorCode := fbPower.ErrorID;
ELSIF fbMoveAbs1.Error THEN
	udnErrorCode := fbMoveAbs1.ErrorID; 
ELSIF fbMoveAbs2.Error THEN
	udnErrorCode := fbMoveAbs2.ErrorID;
ELSIF fbMoveAbs3.Error THEN
	udnErrorCode := fbMoveAbs3.ErrorID;
ELSIF fbHalt.Error THEN
	udnErrorCode := fbHalt.ErrorID;
ELSIF fbReset.Error THEN
	udnErrorCode := fbReset.ErrorID;
ELSIF fbJog.Error THEN
	udnErrorCode := fbJog.ErrorID;
ELSIF fbMoveRel.Error THEN
	udnErrorCode := fbMoveRel.ErrorID;
ELSIF fbMoveVelo.Error THEN
	udnErrorCode := fbMoveVelo.ErrorID;
ELSIF fbMoveModulo.Error THEN
	udnErrorCode := fbMoveModulo.ErrorID;
END_IF

(*Check for Nc error*)
IF NOT bFbError AND Axis.NcToPlc.ErrorCode <> 0 THEN
	bNcError := TRUE;
ELSE 
	bNcError := FALSE;
END_IF

(*Get Nc error code*)
IF bNcError THEN
	udnErrorCode := Axis.NcToPlc.ErrorCode;
END_IF

(*Write error and code*)
bError := bNcError OR bFbError;
IF NOT bError THEN
	udnErrorCode := 0;
END_IF
END_METHOD

METHOD mEventHandler
VAR_INPUT
	Error:						BOOL;
	ErrorCode: 					UDINT;
END_VAR
VAR_INST 
	rtrigError:					R_TRIG;
	rtrigConfirmError:			R_TRIG;
	rtrigClearError:			R_TRIG;
	bAddListener:				BOOL;
	ITcArguments:				I_TcArguments;
END_VAR
(*WRITE*)
	rtrigError(CLK := Error);
	rtrigConfirmError(CLK := bAckError);
	rtrigClearError(CLK := bClearError);
	
	(* Event: Axis generic error *)
	IF rtrigError.Q THEN
		fbTcAlarm_Error.CreateEx(stSeiEvents.Axis_Generic_Error, TRUE, 0);
		fbTcAlarm_Error.ipArguments.Clear().AddUDInt(Axis.NcToPlc.AxisId);
		fbTcAlarm_Error.ipArguments.Clear().AddUDInt(udnErrorCode);	//Does this work?
		fbTcAlarm_Error.Raise(0);
	END_IF
		
	
	(* Event: confirm error *)
	IF rtrigConfirmError.Q THEN
		fbTcAlarm_Error.Confirm(0);
		bAckError := FALSE;
	END_IF
	
	(* Event: clear error *)
	IF rtrigClearError.Q THEN
		fbTcAlarm_Error.Clear(0, TRUE);
	END_IF

(*READ*)
	fbAlarmListener.Execute();
	IF bAddListener THEN
		bAddListener := FALSE;
		fbAlarmListener.Subscribe(0,0);
	END_IF
	
	IF fbAlarmListener.pAlarmConfirmed THEN
		bErrorConfirmed := TRUE;
	END_IF
END_METHOD

METHOD mManualAxisControl : BOOL
VAR_IN_OUT 
	bManualReset:				BOOL;
	bManualPowerOff:			BOOL;
	bManualInit:				BOOL;
END_VAR
VAR_INPUT
	stJogParams:				ST_JOG_PARAMS;
END_VAR
(*
	This method allows for manual control of the axis via input commands
*)
(* Jog Axis *)
IF NOT bManualInit AND NOT bManualReset AND NOT bManualPowerOff THEN
	Axis_Jog(JogParams:= stJogParams);
END_IF
(* Reset Axis *)
IF bManualReset AND NOT bManualInit AND NOT bManualPowerOff THEN
	IF Reset(TRUE) THEN
		Reset(FALSE);
		bManualReset := FALSE;
	END_IF
END_IF
(* Power Off Axis *)
IF bManualPowerOff AND NOT bManualInit AND NOT bManualReset THEN
	IF Axis_PowerOff(TRUE) THEN
		Axis_PowerOff(FALSE);
		bManualPowerOff := FALSE;
	END_IF
END_IF
(* Re-Initialize Axis*) 
IF bManualInit AND NOT bManualPowerOff AND NOT bManualReset THEN
	IF Initialize(TRUE) THEN
		Initialize(FALSE);
		bManualInit := FALSE;
	END_IF
END_IF
END_METHOD

METHOD MoveAbs : BOOL
VAR_INPUT
	Execute:			BOOL;
	MotionParams:		ST_MOTION_PARAMS;
END_VAR
VAR_INST
	State :				INT;
END_VAR
rtrigExecute(CLK := Execute);
CASE State OF
	0: //Execute
		IF rtrigExecute.Q THEN
			MoveAbs := FALSE;
			bDidMoveAbs := FALSE;
			State := 10;
		END_IF
	10: //Move 
		fbMoveAbs1.Position:= MotionParams.TargetPos; 
		fbMoveAbs1.Velocity:= MotionParams.TargetVel; 
		fbMoveAbs1.Acceleration:= MotionParams.TargetAccel; 
		fbMoveAbs1.Deceleration:= MotionParams.TargetDecel;
		fbMoveAbs1.Jerk:= MotionParams.Jerk;
		fbMoveAbs1.Execute:= TRUE;  
		IF fbMoveAbs1.Done THEN
			fbMoveAbs1.Execute:= FALSE;
			MoveAbs := TRUE;
			bDidMoveAbs := TRUE;		
			State := 0;
		END_IF
END_CASE
END_METHOD

METHOD MoveAbsBuffered : BOOL
VAR_INPUT
	Execute :				BOOL;
	MotionParamsP1 :		ST_MOTION_PARAMS;	//Motion 1 paramters (MC_Buffered must be used for BufferMode)
	MotionParamsP2 :		ST_MOTION_PARAMS;	//Motion 2 paramters (MC_BlendingNext, High, Low, Previous )
END_VAR
VAR_INST
	State :					INT;
END_VAR
rtrigExecute(CLK := Execute);
CASE State OF
	0: //Execute
		IF rtrigExecute.Q THEN
			MoveAbsBuffered := FALSE;
			State := 10;
		END_IF	
	10: //Execute motion 1 
		fbMoveAbs1.Execute := TRUE;
		fbMoveAbs1.Position := MotionParamsP1.TargetPos;
		fbMoveAbs1.Velocity := MotionParamsP1.TargetVel; 
		fbMoveAbs1.Acceleration := MotionParamsP1.TargetAccel; 
		fbMoveAbs1.Deceleration := MotionParamsP1.TargetAccel; 
		fbMoveAbs1.Jerk := MotionParamsP1.Jerk;
		fbMoveAbs1.BufferMode := MotionParamsP1.BufferMode;
		IF fbMoveAbs1.Active THEN
			fbMoveAbs1.Execute := FALSE;
			State := 20;
		ELSIF NOT Execute THEN
			State := 0;;			
		END_IF 
	20: //Execute motion 2
		fbMoveAbs2.Execute := TRUE;
		fbMoveAbs2.Position := MotionParamsP2.TargetPos;
		fbMoveAbs2.Velocity := MotionParamsP2.TargetVel; 
		fbMoveAbs2.Acceleration := MotionParamsP2.TargetAccel; 
		fbMoveAbs2.Deceleration := MotionParamsP2.TargetAccel; 
		fbMoveAbs2.Jerk := MotionParamsP2.Jerk;
		fbMoveAbs2.BufferMode := MotionParamsP2.BufferMode;
		IF fbMoveAbs2.Done THEN
			fbMoveAbs2.Execute := FALSE;
			State := 30;
		ELSIF NOT Execute THEN
			State := 0;;			
		END_IF
	30: //Check busy output for completion 
		IF NOT fbMoveAbs1.Busy AND NOT fbMoveAbs2.Busy THEN
			MoveAbsBuffered := TRUE;
			State := 0;
		END_IF
END_CASE
END_METHOD

METHOD MoveAbsBuffered3Pos : BOOL
VAR_INPUT
	Execute :				BOOL;
	MotionParamsP1 :		ST_MOTION_PARAMS;	//Motion 1 paramters (MC_Buffered must be used for BufferMode)
	MotionParamsP2 :		ST_MOTION_PARAMS;	//Motion 2 paramters (MC_BlendingNext, High, Low, Previous )
	MotionParamsP3 :		ST_MOTION_PARAMS;	//Motion 3 paramters (MC_BlendingNext, High, Low, Previous )
END_VAR
VAR_INST
	State :					INT;
END_VAR
rtrigExecute(CLK := Execute);
CASE State OF
	0: //Execute
		IF rtrigExecute.Q THEN
			MoveAbsBuffered3Pos := FALSE;
			State := 10;
		END_IF	
	10: //Execute motion 1 
		fbMoveAbs1.Execute := TRUE;
		fbMoveAbs1.Position := MotionParamsP1.TargetPos;
		fbMoveAbs1.Velocity := MotionParamsP1.TargetVel; 
		fbMoveAbs1.Acceleration := MotionParamsP1.TargetAccel; 
		fbMoveAbs1.Deceleration := MotionParamsP1.TargetAccel; 
		fbMoveAbs1.Jerk := MotionParamsP1.Jerk;
		fbMoveAbs1.BufferMode := MotionParamsP1.BufferMode;
		IF fbMoveAbs1.Active THEN
			fbMoveAbs1.Execute := FALSE;
			State := 20;
		ELSIF NOT Execute THEN
			State := 0;;			
		END_IF 
	20: //Execute motion 2
		fbMoveAbs2.Execute := TRUE;
		fbMoveAbs2.Position := MotionParamsP2.TargetPos;
		fbMoveAbs2.Velocity := MotionParamsP2.TargetVel; 
		fbMoveAbs2.Acceleration := MotionParamsP2.TargetAccel; 
		fbMoveAbs2.Deceleration := MotionParamsP2.TargetAccel; 
		fbMoveAbs2.Jerk := MotionParamsP2.Jerk;
		fbMoveAbs2.BufferMode := MotionParamsP2.BufferMode;
		IF fbMoveAbs2.Active THEN
			fbMoveAbs2.Execute := FALSE;
			State := 30;
		ELSIF NOT Execute THEN
			State := 0;
		END_IF
	30:	//Execute motion 2
		fbMoveAbs3.Execute := TRUE;
		fbMoveAbs3.Position := MotionParamsP3.TargetPos;
		fbMoveAbs3.Velocity := MotionParamsP3.TargetVel; 
		fbMoveAbs3.Acceleration := MotionParamsP3.TargetAccel; 
		fbMoveAbs3.Deceleration := MotionParamsP3.TargetAccel; 
		fbMoveAbs3.Jerk := MotionParamsP3.Jerk;
		fbMoveAbs3.BufferMode := MotionParamsP3.BufferMode;
		IF fbMoveAbs3.Done THEN
			fbMoveAbs3.Execute := FALSE;
			State := 40;
		ELSIF NOT Execute THEN
			State := 0;;			
		END_IF
	40: //Check busy output for completion 
		IF NOT fbMoveAbs1.Busy AND NOT fbMoveAbs2.Busy AND NOT fbMoveAbs3.Busy THEN
			MoveAbsBuffered3Pos := TRUE;
			State := 0;
		END_IF
END_CASE
END_METHOD

METHOD PUBLIC MoveVelo : BOOL
VAR_INPUT
	Execute :				BOOL;
	MotionParams:			ST_MOTION_PARAMS;
END_VAR
VAR_INST
	State:					INT;
END_VAR
rtrigExecute(CLK := Execute);
CASE State OF 
	0:	// Execute
		IF rtrigExecute.Q THEN
			MoveVelo := FALSE;
			bDidMoveVelo := FALSE;
			State := 10;
		END_IF
	10://Move Velocity
			fbMoveVelo.Execute:= TRUE;
			fbMoveVelo.Velocity:= MotionParams.TargetVel; 
			fbMoveVelo.Acceleration:= MotionParams.TargetAccel; 
			fbMoveVelo.Deceleration:= MotionParams.TargetDecel; 
			fbMoveVelo.Jerk:= MotionParams.Jerk; 
			fbMoveVelo.Direction:= MotionParams.Direction; 
		IF fbMoveVelo.InVelocity THEN
			fbMoveVelo.Execute:= FALSE;
			MoveVelo := TRUE;
			bDidMoveVelo := TRUE;
			State := 0;
		END_IF
END_CASE
END_METHOD

METHOD mStopWithOverride : BOOL
VAR_INPUT
	udnOverride			:	UDINT;
	bUseOverrideOK		:	BOOL;	//Signal is true when override is used, otherwise zero.
END_VAR
IF bUseOverrideOK AND GVL.bCurrentIsZero THEN
	SetAxisOverride(Override := udnOverride);
ELSE
	SetAxisOverride(Override := 0);
END_IF
END_METHOD

PROPERTY pAckError : BOOL
GET
END_GET
SET
END_SET
END_PROPERTY

METHOD Pause : BOOL
Pause := FALSE;
fbPower.Override := 0;
Pause := TRUE;
END_METHOD

PROPERTY pClearError : BOOL
SET
END_SET
END_PROPERTY

PROPERTY pError : BOOL
GET
pError := bError;
END_GET
SET
END_SET
END_PROPERTY

PROPERTY pErrorCleared : BOOL
GET
END_GET
END_PROPERTY

PROPERTY pErrorCode : UDINT
GET
pErrorCode := udnErrorCode;
END_GET
SET
END_SET
END_PROPERTY

PROPERTY pErrorConfirmed : BOOL
GET
END_GET
END_PROPERTY

PROPERTY pErrorDescription : T_MaxString
GET
END_GET
SET
END_SET
END_PROPERTY

PROPERTY pIsMoving : BOOL
GET
pIsMoving := fbMoveAbs1.Busy OR fbMoveAbs2.Busy OR fbMoveAbs3.Busy OR fbMoveModulo.Busy OR fbMoveVelo.Busy OR fbMoveRel.Busy OR fbJog.Busy;
END_GET
END_PROPERTY

METHOD Ref : BOOL
VAR_INPUT
	Execute:	BOOL;
END_VAR
VAR_INST 
	State:		INT;
END_VAR
rtrigExecute(CLK := Execute);
CASE State OF	
	0: //Execute 
		IF rtrigExecute.Q THEN
			bDidRef := FALSE;
			Ref := FALSE;
			State := 10;
		END_IF
	10: //Reference
		Ref := TRUE;
		bDidRef := TRUE;
		IF Ref THEN
			State := 0;
		END_IF 
END_CASE
END_METHOD

METHOD Reset : BOOL
VAR_INPUT
	Execute:		BOOL;
END_VAR
VAR_INST
	State:			INT;
	rtrigReset:		R_TRIG;
END_VAR
rtrigReset(CLK := Execute);
CASE State OF
	0: //Execute
		IF rtrigReset.Q THEN
			Reset := FALSE;
			bDidReset := FALSE;
			State := 10;
		END_IF
	10: //Reset 
		fbReset.Execute:= TRUE;
		IF fbReset.Done THEN
			fbReset.Execute := FALSE;
			bDidReset := TRUE;
			Reset := TRUE;
			State := 0;
		END_IF	
END_CASE
END_METHOD

METHOD Resume : BOOL
VAR_INPUT
	ResumeOverride: LREAL;
END_VAR
Resume := FALSE;
fbPower.Override := ResumeOverride;
Resume := TRUE;
END_METHOD

METHOD SetAxisOverride
VAR_INPUT
	Override:				UDINT;						//Set value from 0-100%
END_VAR
(*
	This method passes an override value to the NC 
*)
fbPower.Override := Override;
END_METHOD

PROPERTY Status : BOOL
GET
Status := fbPower.Status;
END_GET
END_PROPERTY

METHOD Stop : BOOL
VAR_INPUT
	Execute:			BOOL;
	MotionParams:		ST_MOTION_PARAMS;
END_VAR
VAR_INST
	State:				INT;
	rtrigHalt:			R_TRIG;
END_VAR
rtrigHalt(CLK := Execute);
CASE State OF 
	0:	//Execute
		IF Execute THEN
			Stop := FALSE;
			State := 10;
		END_IF
	10://Halt 
		fbStop.Deceleration:= MotionParams.TargetDecel; 
		fbStop.Jerk:= MotionParams.Jerk; 
		fbStop.Execute:= TRUE;
END_CASE
END_METHOD

END_FUNCTION_BLOCK

// ---- POUs/00_Shared/FB_AlarmListener.TcPOU
(*
	The function block serves as the basic implementation of an event listener.
	New messages and state changes of alarms can be recognized through the overwriting of the event-driven
	methods.
*)
FUNCTION_BLOCK FB_AlarmListener EXTENDS FB_ListenerBase2
VAR
(*POUs*)
	fbRequestEventText:			FB_RequestEventText;
(*Property vars*)
	udnLastEventID: 			UDINT;
	ulnLastEventTimeStamp: 		ULINT;
	sLastEventText: 			STRING;
	bReqEventText: 				BOOL;
	bAlarmRaised:				BOOL;
	bAlarmConfirmed:			BOOL;
	bAlarmCleared:				BOOL;
END_VAR

METHOD Execute : HRESULT
VAR_INPUT
END_VAR
Execute := SUPER^.Execute(); //retrieve events

//retrieve the text of a message
IF 	bReqEventText AND fbRequestEventText.bError THEN 
	sLastEventText := 'Error';
	bReqEventText := FALSE; 
ELSIF bReqEventText AND NOT  fbRequestEventText.bBusy THEN
	fbRequestEventText.GetString(sLastEventText, SIZEOF(sLastEventText));
	bReqEventText := FALSE;
END_IF
END_METHOD

METHOD OnAlarmCleared : HRESULT
VAR_INPUT
	fbEvent:	REFERENCE TO FB_TcEvent;
END_VAR
//Get alarm ID 
udnLastEventID := fbEvent.nEventId;
//Get alarm time stamp
ulnLastEventTimeStamp := fbEvent.nTimestamp;
//Send request to get alarm text 
fbRequestEventText.Request(eventClass := fbEvent.EventClass, nEventId := fbEvent.nEventId, nLangId := 1033, ipArgs := fbEvent.ipArguments);
bReqEventText := TRUE;
//Validate alarm cleared
bAlarmCleared := TRUE;
END_METHOD

METHOD OnAlarmConfirmed : HRESULT
VAR_INPUT
	fbEvent:	REFERENCE TO FB_TcEvent;
END_VAR
//Get alarm ID 
udnLastEventID := fbEvent.nEventId;
//Get alarm time stamp
ulnLastEventTimeStamp := fbEvent.nTimestamp;
//Send request to get alarm text 
fbRequestEventText.Request(eventClass := fbEvent.EventClass, nEventId := fbEvent.nEventId, nLangId := 1033, ipArgs := fbEvent.ipArguments);
bReqEventText := TRUE;
//Validate alarm confirmed
bAlarmConfirmed := TRUE;
END_METHOD

METHOD OnAlarmRaised : HRESULT
VAR_INPUT
	fbEvent:	REFERENCE TO FB_TcEvent;
END_VAR
//Get alarm ID 
udnLastEventID := fbEvent.nEventId;
//Get alarm time stamp
ulnLastEventTimeStamp := fbEvent.nTimestamp;
//Send request to get alarm text 
fbRequestEventText.Request(eventClass := fbEvent.EventClass, nEventId := fbEvent.nEventId, nLangId := 1033, ipArgs := fbEvent.ipArguments);
bReqEventText := TRUE;
//Validate alarm raised
bAlarmRaised := TRUE;
END_METHOD

PROPERTY pAlarmCleared : BOOL
GET
pAlarmCleared := bAlarmCleared;
END_GET
SET
bAlarmCleared := pAlarmCleared;
END_SET
END_PROPERTY

PROPERTY pAlarmConfirmed : BOOL
GET
pAlarmConfirmed := bAlarmConfirmed;
END_GET
SET
bAlarmConfirmed := pAlarmConfirmed;
END_SET
END_PROPERTY

PROPERTY pAlarmRaised : BOOL
GET
pAlarmRaised := bAlarmRaised;
END_GET
SET
bAlarmRaised := pAlarmRaised;
END_SET
END_PROPERTY

PROPERTY pLastEventID : udint
GET
pLastEventID := udnLastEventID;
END_GET
END_PROPERTY

PROPERTY pLastEventText : string
GET
pLastEventText := sLastEventText;
END_GET
END_PROPERTY

PROPERTY pLastEventTimeStamp : ulint
GET
pLastEventTimeStamp := ulnLastEventTimeStamp;
END_GET
END_PROPERTY

END_FUNCTION_BLOCK

// ---- POUs/FB_Light.TcPOU
FUNCTION_BLOCK FB_Light

VAR
	bColor1 AT %Q* : BYTE := 1;
	bColor2 AT %Q* : BYTE := 0;
	bFlashRate AT %Q* : BYTE := 1;
	bColor1Intensity AT %Q* : BYTE := 1;
	bColor2Intensity AT %Q* : BYTE := 1;
	bAudibleMode AT %Q* : BYTE := 0;
	bAnimationMode AT %Q* : BYTE := 1;
	bRotationalMode AT %Q* : BYTE := 0;

	tonTimerDelay1 : TON := (PT := T#500MS);
	tonTimerDelay2 : TON := (PT := T#500MS);
	
	nColorIndex : BYTE := 0;
END_VAR

METHOD mActivate : BOOL

VAR_INPUT
	inputVariable : BOOL;
END_VAR

VAR_INST
	localVar : BOOL;
END_VAR
localVar := inputVariable;

IF localVar THEN
	bAnimationMode := 1;
ELSE
	bAnimationMode := 0;
END_IF
END_METHOD

METHOD mCheckStatus : BOOL
VAR_INPUT
	bInputStatus : BOOL;
END_VAR



VAR
	tonTimeDelay : TON := (PT := T#4S);
END_VAR
IF bInputStatus THEN
	bColor1 := 0;
ELSE
	bColor1 := 1;
END_IF
END_METHOD

METHOD mFillArray : BOOL

VAR_INPUT
	//
END_VAR

VAR
	nIndex : INT := 1;
END_VAR

//FOR nIndex := 1 TO SIZEOF(aColors) DO
	//aColors[nIndex] := nIndex;
//END_FOR
END_METHOD

METHOD mLightDelay : BOOL

VAR_INPUT
	bInputState : BOOL; // case reset button from input
END_VAR

VAR_INST
	nCaseState : INT := 1;
	trigger : R_TRIG;
	
END_VAR
CASE nCaseState OF
	1:
		tonTimerDelay1(IN := TRUE);	
		IF tonTimerDelay1.Q THEN
			bColor1 := 1; // RED
			tonTimerDelay1(IN := FALSE);
			nCaseState := 2;
		END_IF

	2:
		tonTimerDelay2(IN := TRUE);
		IF tonTimerDelay2.Q THEN
			bColor1 := 0; // GREEN
			tonTimerDelay2(IN := FALSE);
			nCaseState := 1;
		END_IF
	
END_CASE
END_METHOD

METHOD mLightSpectrum : BOOL

VAR_INPUT
	//bInputState : BOOL; // case reset button from input
END_VAR

VAR_INST
	nCaseState : INT := 1;
	trigger : R_TRIG;
	
END_VAR
CASE nCaseState OF
	1:
		tonTimerDelay1(IN := TRUE);	
		IF tonTimerDelay1.Q THEN
			IF nColorIndex > 12 THEN
				nColorIndex := 0;
			END_IF
			bColor1 := nColorIndex;
			nColorIndex := nColorIndex + 1;
			
			tonTimerDelay1(IN := FALSE);
			nCaseState := 2;
		END_IF

	2:
		tonTimerDelay2(IN := TRUE);
		IF tonTimerDelay2.Q THEN
			IF nColorIndex > 12 THEN
				nColorIndex := 0;
			END_IF
			bColor1 := nColorIndex;
			nColorIndex := nColorIndex + 1;

			tonTimerDelay2(IN := FALSE);
			nCaseState := 1;
		END_IF
	
END_CASE
END_METHOD

METHOD mSetAnimation : BOOL

VAR_INPUT
	bInputValue : BYTE;
END_VAR
bAnimationMode := bInputValue;
END_METHOD

METHOD mSetColor : BOOL

VAR_INPUT
	nInputNumber : INT;
END_VAR

bColor1 := INT_TO_BYTE(nInputNumber);
END_METHOD

END_FUNCTION_BLOCK

// ---- POUs/FB_Button.TcPOU
FUNCTION_BLOCK FB_Button

VAR
	byButtonInput AT %I* : BIT;
	byButtonLight AT %Q* : BIT;
END_VAR

METHOD mButtonLight : BOOL

VAR_INPUT
	//byButtonInput : BYTE;
END_VAR

IF byButtonInput THEN
	byButtonLight := TRUE;

ELSE
	byButtonLight := FALSE;
END_IF
END_METHOD

END_FUNCTION_BLOCK
